{attribute 'GeneratedUsingTerminal: EL3681-0000-0018'}
{attribute addProperty BoxType "EL3681-0000-0018"}
{attribute addProperty Id "ControlAT %Q*Control_18D542D94"}
{attribute addProperty CRC "706248645"}
{attribute addProperty Size "4"}
TYPE SAI_Range_2A187FC5 EXTENDS OutputBase_10CEE7DE :
STRUCT
	{attribute addProperty Name "Control"}
	Control AT %Q* : Control_18D542D9;
END_STRUCT
END_TYPE

(* stored: Version 1.2.0.0, ProductVersion 3.1.4024.9
   DUT SAI_Range_2A187FC5: Id {c13a0a74-2964-4996-891c-c4836e5c1ef9} *)
